// TIA Portal V17 export
// export: Created 2025-03-10T12:17:22.0726893Z, ExportSetting WithDefaults, DisplayName Totally Integrated Automation Portal, DisplayVersion V17 Update 8, DisplayName TIA Portal Openness, DisplayVersion V17 Update 8, DisplayName TIA Portal Version Control Interface, DisplayVersion V17, DisplayName SINAMICS Startdrive Advanced, DisplayVersion V17 SP2, DisplayName SINAMICS Startdrive G110M, G120, G120C, G120D, G120P, G115D, DisplayVersion V17 SP2, DisplayName SINAMICS Startdrive G130, G150, S120, S150, SINAMICS MV, S210, DisplayVersion V17 SP2, DisplayName STEP 7 Professional, DisplayVersion V17 Update 8, DisplayName SINUMERIK ONE STEP 7 Toolbox, DisplayVersion V17 Update 12, DisplayName SINUMERIK 840D sl STEP 7 Toolbox, DisplayVersion V17 Update 12, DisplayName STEP 7 Safety, DisplayVersion V17 Update 6, DisplayName WinCC Advanced, DisplayVersion V17 Update 8
DATA_BLOCK "DB7230_ENABLE_OPTIONS"   // DB7230
{ S7_Optimized_Access := 'FALSE'; DB_Accessible_From_OPC_UA := 'FALSE' }
AUTHOR : ETXETAR
VERSION : 1.0
// stored: AutoNumber false, DBAccessibleFromOPCUA false, DBAccessibleFromWebserver true, IsOnlyStoredInLoadMemory false, IsWriteProtectedInAS false
   VAR RETAIN
      ENABLE_REQUEST : Array[1..200] of Bool;   // Monitor Enable Request / ENABLE REQUEST
      DISABLE_REQUEST : Array[1..200] of Bool;   // Monitor Disable Request / DISABLE REQUEST
      MACHINE_STRUCTURE_STATUS : Array[1..100] of Bool;   // Monitor Status / STATUS
      MACHINE_DEVICE_STATUS : Array[1..100] of Bool;   // Monitor Status / STATUS
      HMI_MACHINE_STRUCTURE_ENABLE_REQUEST : Bool;   // HMI MACHINE STRUCTURE ENABLE REQUEST
      HMI_MACHINE_STRUCTURE_DISABLE_REQUEST : Bool;   // HMI MACHINE STRUCTURE DISABLE REQUEST
      HMI_MACHINE_DEVICE_ENABLE_REQUEST : Bool;   // HMI MACHINE DEVICE ENABLE REQUEST
      HMI_MACHINE_DEVICE_DISABLE_REQUEST : Bool;   // HMI MACHINE DEVICE DISABLE REQUEST
      HMI_MACHINE_STRUCTURE_TABLE_LINE : Byte := 16#1;   // HMI MACHINE STRUCTURE TABLE LINE
      HMI_MACHINE_DEVICE_TABLE_LINE : Byte := 16#1;   // HMI MACHINE DEVICE TABLE LINE
   END_VAR
BEGIN
END_DATA_BLOCK
